Omron Sysmac Studio project FORLOOP (Sysmac Studio 1.56.0.64011, StandardProject)

# Controller new_Controller_0: NJ501-1500 version 1.64
Units and slaves: Power Supply : NJ-Px3001; CPU : NJ501-1500
Task PrimaryTask (priority 4, period or condition 1000): Program0

VAR_GLOBAL
    Board : ARRAY[1..2,1..10] OF INT;
    Even : INT := 0;
    Odd : INT := 0;
    EvenArray : ARRAY[1..10] OF INT := [2, 4, 6, 8, 10, 12, 14, 16, 18, 20];
    OddArray : ARRAY[1..10] OF INT := [10, 9, 8, 7, 6, 5, 4, 3, 2, 1];
END_VAR

PROGRAM Program0
VAR_EXTERNAL
    Board : ARRAY[1..2,1..10] OF INT;
    Even : INT;
    EvenArray : ARRAY[1..10] OF INT;
    OddArray : ARRAY[1..10] OF INT;
END_VAR

(* Section Section0: ladder, written here as Structured Text *)

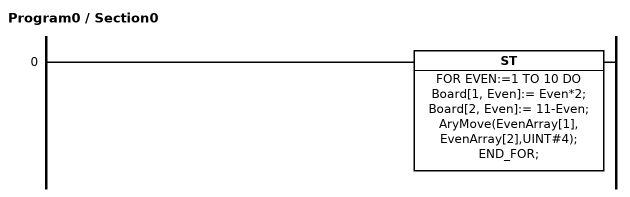
(* Rung 0 *)
FOR EVEN:=1 TO 10 DO
	Board[1, Even]:= Even*2;
	Board[2, Even]:= 11-Even;
	AryMove(EvenArray[1],EvenArray[2],UINT#4);
END_FOR;
END_PROGRAM